PROGRAM PRG_HV_ILK
VAR
END_VAR

(*High Voltage Saftey Loop*)
IF DREAM_MC_GHC.M_IsCh1Selected() THEN
    bHighVoltageSafteyLoopEnable := (DREAM_MC_GHC.IG_CH1.rPRESS <= fHighVoltageMinPressure) AND DREAM_MC_GHC.IG_CH1.xPRESS_OK;
ELSIF DREAM_MC_GHC.M_IsCh2Selected() THEN
    bHighVoltageSafteyLoopEnable := (DREAM_MC_GHC.IG_CH2.rPRESS <= fHighVoltageMinPressure) AND DREAM_MC_GHC.IG_CH2.xPRESS_OK;
ELSE
    bHighVoltageSafteyLoopEnable := FALSE;
END_IF

END_PROGRAM

(* stored: Version 1.1.0.1, ProductVersion 3.1.4024.12
   POU PRG_HV_ILK: Id {d0f59b88-3cfc-41d8-b70c-ef6b66a977a9}, SpecialFunc None *)
